// Parses a double value.
FUNCTION F_ParseDouble : HRESULT
VAR_IN_OUT CONSTANT
    aBuffer : ARRAY [*] OF BYTE;   
END_VAR
VAR_IN_OUT
    stState : ST_ParserInternalState;
END_VAR
VAR_OUTPUT
    fValue : LREAL;
END_VAR
VAR CONSTANT
    cLength : UDINT := SIZEOF(fValue);
END_VAR
VAR
    fTmp : LREAL;
END_VAR


F_ParseDouble := S_OK;

IF stState.nBufferSize - stState.nBufferPos < cLength THEN
    F_ParseDouble := stState.eParserErrorCode := E_ParserErrorCode.TruncatedMessage;
    stState.bError := TRUE;
    RETURN;
END_IF

MEMCPY(destAddr:= ADR(fTmp), srcAddr:= ADR(aBuffer[stState.nBufferPos]), n:= cLength);
stState.nBufferPos := stState.nBufferPos + cLength;

{warning 'TODO: Check for endianess?'}
fValue := fTmp;

END_FUNCTION

(* stored: Version 1.1.0.1
   POU F_ParseDouble: Id {24606ab3-3eb3-493e-9ecb-d98469f178b3}, SpecialFunc None *)
